FUNCTION_BLOCK GantryPick
VAR_INPUT
	En: BOOL;
	PickStation: INT;
	PickPosition: INT;
END_VAR
VAR_OUTPUT
	Done: BOOL;
	Executing: BOOL;
	Waiting: BOOL;
	Error: BOOL;
	Progress: INT;
END_VAR
VAR_IN_OUT
	Data:CommunicationData;
END_VAR
VAR
END_VAR


IF En THEN

	// Auto sequence pick pallet
	CASE Progress OF
		0:	//Clear old order
			Data.PickStation := 0;
			Data.PickPosition := 0;
			Progress := 10;

		10:	//Start gantry robot auto squence
			IF Data.Auto AND PickStation > 0 AND  PickStation <= 4 AND PickPosition > 0 AND PickPosition <= 9 THEN
				Data.PickStation := PickStation;
				Data.PickPosition := PickPosition;
				Executing := FALSE;
				Waiting := FALSE;
				Error := FALSE;
				Progress := 30;
			ELSE
				Executing := FALSE;
				Waiting := FALSE;
				Error := TRUE;
			END_IF

		30: // Check acknowledge from GantryRobot
			IF Data.AckPickStation = PickStation AND Data.AckPickPosition = PickPosition THEN
				Executing := TRUE;
				Waiting := FALSE;
				Error := FALSE;
				Progress := 50;
			ELSE
				Executing := FALSE;
				Waiting := TRUE;
				Error := NOT Data.Auto;
			END_IF
			
		50: // Wait for gantry auto squence ready and clear order	
			IF Data.AckPickStation = 0 AND Data.AckPickPosition = 0 THEN
				Data.PickStation := 0;
				Data.PickPosition := 0;
				Executing := FALSE;
				Waiting := FALSE;
				Error := FALSE;
				Progress := 100;
			ELSE
				Executing := TRUE;
				Waiting := FALSE;
				Error := NOT Data.Auto;
			END_IF
		
		100: // Operation done
			Done := TRUE;
	END_CASE

ELSE //En
	IF Progress > 0 THEN
		Data.PickStation := 0;
		Data.PickPosition := 0;	
	END_IF
	Progress := 0;
	Done := FALSE;
	Executing := FALSE;
	Waiting := FALSE;
	Error := FALSE;
END_IF

END_FUNCTION_BLOCK

(* stored: Version 1.1.0.1, ProductVersion 3.1.4022.12
   POU GantryPick: Id {0e6931f0-f20c-44c4-b637-b8cf98b9ec7b}, SpecialFunc None *)
